{attribute 'qualified_only'}
VAR_GLOBAL
	emergency: BOOL;
	iDialogManager : VisuElems.IDialogManager;
	iMessageDialog : VisuElems.IVisualisationDialog;
END_VAR

(* stored: Version 1.1.0.1, ProductVersion 3.1.4024.12
   GVL GVL: Id {4c860135-d774-4f18-9c2d-8709fca93d47} *)
